TYPE T_LongSTRING : STRING(1023);
END_TYPE

(* stored: Version 1.1.0.1
   DUT T_LongSTRING: Id {89b3592c-feec-4798-9abb-2f72ccd8807b} *)
